{attribute 'qualified_only'}
VAR_GLOBAL
	StopButton AT %I* : BOOL;
	EmergencyStopButton AT %I* : BOOL;
	StartButton AT %I* : BOOL;
	ProductDetectedSensor AT %I* : BOOL;
	ConveyorFullSensor AT %I* : BOOL;
	MotorContactor AT %Q* : BOOL;
END_VAR

(* stored: Version 1.1.0.1, ProductVersion 3.1.4024.9
   GVL GVL: Id {aa76d518-5d0c-47e9-a040-3c7a082b4032} *)
